(* CODESYS project canbus.20191014.1.project

Project tree, tasks and I/O mapping:
  Changsha_Xiangji_ARM_Cortex_A9_xilinx_zynq7000_linux : Changsha Xiangji-ARM Cortex A9(xilinx zynq7000)-linux, Changsha Xiangji Hiden Technology Co.Ltd, version 3.5.10.40
    application Application
      libraries: VisuDialogs, * (System); CAA Real Time Clock Extern, 3.5.10.0 (CAA Technical Workgroup); CAA Callback Extern, 3.5.11.0 (CAA Technical Workgroup); CAA Can Low Level Imp Extern, 3.5.11.0 (CAA Technical Workgroup); SysMem, 3.5.12.0 (System); CAA SerialCom, 3.5.12.0 (CAA Technical Workgroup); CAA DTUtil Extern, 3.5.12.0 (CAA Technical Workgroup); SysFile, 3.5.9.0 (System); SysTypes2 Interfaces, * (System); CAA Types Extern, 3.5.13.0 (CAA Technical Workgroup); CAA Can Low Level Extern, 3.5.13.0 (CAA Technical Workgroup); CAA Net Base Services, 3.5.13.0 (CAA Technical Workgroup); Standard, 3.5.13.0 (System); CAA File, 3.5.13.40 (CAA Technical Workgroup)
      task VISU_TASK (cyclic, interval 100 ms, priority 31) calls VisuElems.Visu_Prg
      task task_can (cyclic, interval 4 ms, priority 5) calls prg_can0, prg_can1, prg_test_can
      CAN_COMM/
        program prg_can0 [ST]
        function CAN_Send_MSG [ST]
        program prg_can1 [ST]: can1_get_data1, can1_get_data3, can1_get_data2, can1_set_send_buf
        program prg_test_can [ST]
      visualisation main
      funcs/
    SoftMotion General Axis Pool
    IoDrvMIC7001 : IoDrvMIC7001, Cyber-MI, version 18.11.1
        unmapped channels: Ai00@C16, Ai01@C28, Ai02@C17, Ai03@C29, Ai04@C30, Ai05@C19, Ai06@C31, Ai07@C20, Ai08@C18, Ai09@D18, Ai10@D20, Ai11@D31, Ai12@D19, Ai13@D30, Ai14@D29, Ai15@D17, Ai16@D28, Ai17@D16, Ai18-Do00@C25, Ai19-Do01@C24, Ai20-Do02@C13, Ai21-Do03@C01, Ai22-Do04@C03, Ai23-Do05@C04, Ai24-Do06@C05, Ai25-Do07@C06, Ai26-Do08@C08, Ai27-Do09@C09, Ai28-Do10@C10, Ai29-Do11@C11, Ai30-Do12@D34, Ai31-Do13@D35, Ai32-Do14@D23, Ai33-Do15@D12, Ai34-Do16@D10, Ai35-Do17@D09, Ai36-Do18@D08, Ai37-Do19@D07, Ai38-Do20@D05, Ai39-Do21@D04,
          Ai40-Do22@D03, Ai41-Do23@D02, Ai42-Do24@C23, Ai43-Do25@C35, Ai44-Do26@D24, Ai45-Do27@D13, Ai46-Ao00@C22, Ai47-Ao01@D14, Ai48_Pi02, Ai49_Out5V, Ai50_VCC, Ai51_VCC_L, Ai52_VCC_R, Ai53_Pwm-i0, Ai54_Pwm-i1, Ai55_Pwm-i2, Ai56_Pwm-i3, Ai57_CPU-T, Ai58_G-x, Ai59_G-y, Ai60_G-z, Ai61-reserved, Ai62-IO-cntr, Ai63-CDS-cntr, Di00-Ai00@C16, Di01-Ai01@C28, Di02-Ai02@C17, Di03-Ai03@C29, Di04-Ai04@C30, Di05-Ai05@C19, Di06-Ai06@C31, Di07-Ai07@C20, Di08-Ai08@C18, Di09-Ai09@D18, Di10-Ai10@D20, Di11-Ai11@D31, Di12-Ai12@D19, Di13-Ai13@D30, Di14-Ai14@D29, Di15-Ai15@D17,
          Di16-Ai16@D28, Di17-Ai17@D16, Di18-Ai18@C25, Di19-Ai19@C24, Di20-Ai20@C13, Di21-Ai21@C01, Di22-Ai22@C03, Di23-Ai23@C04, Di24-Ai24@C05, Di25-Ai25@C06, Di26-Ai26@C08, Di27-Ai27@C09, Di28-Ai28@C10, Di29-Ai29@C11, Di30-Ai30@D34, Di31-Ai31@D35, Di32-Ai32@D23, Di33-Ai33@D12, Di34-Ai34@D10, Di35-Ai35@D09, Di36-Ai36@D08, Di37-Ai37@D07, Di38-Ai38@D05, Di39-Ai39@D04, Di40-Ai40@D03, Di41-Ai41@D02, Di42-Ai42@C23, Di43-Ai43@C35, Di44-Ai44@D24, Di45-Ai45@D13, Di46-Ai46@C22, Di47-Ai47@D14, Di48-Pi00@C15, Di49-Pi01@C14, Di50-Pi02@D22, Di51-Pi03@D21, Di52-reserved, Di53-reserved, Di54-reserved, Di55-reserved,
          Di56-reserved, Di57-reserved, Di58-reserved, Di59-reserved, Di60-reserved, Di61-reserved, Di62-reserved, Di63-reserved, Pi00-Di48@C15, Pi01-Di49@C14, Pi02-Di50@D22, Pi03-Di51@D21, Do00-Ai18@C25, Do01-Ai19@C24, Do02-Ai20@C13, Do03-Ai21@C01, Do04-Ai22@C03, Do05-Ai23@C04, Do06-Ai24@C05, Do07-Ai25@C06, Do08-Ai26@C08, Do09-Ai27@C09, Do10-Ai28@C10, Do11-Ai29@C11, Do12-Ai30@D34, Do13-Ai31@D35, Do14-Ai32@D23, Do15-Ai33@D12, Do16-Ai34@D10, Do17-Ai35@D09, Do18-Ai36@D08, Do19-Ai37@D07, Do20-Ai38@D05, Do21-Ai39@D04, Do22-Ai40@D03, Do23-Ai41@D02, Do24-Ai42@C23, Do25-Ai43@C35, Do26-Ai44@D24, Do27-Ai45@D13,
          Do28-Pwmi00@C33, Do29-Pwmi01@C34, Do30-Pwmi02@D25, Do31-Pwmi03@D26, PWM00@C25, PWM01@C24, PWM02@C13, PWM03@C01, PWM04@C03, PWM05@C04, PWM06@C05, PWM07@C06, PWM08@C08, PWM09@C09, PWM10@C10, PWM11@C11, PWM12@D34, PWM13@D35, PWM14@D23, PWM15@D12, PWM16@D10, PWM17@D09, PWM18@D08, PWM19@D07, PWM20@D05, PWM21@D04, PWM22@D03, PWM23@D02, PWM24@C23, PWM25@C35, PWM26@D24, PWM27@D13, PWM28-Pwmi00@C33, PWM29-Pwmi01@C34, PWM30-Pwmi02@D25, PWM31-Pwmi03@D26, PWM_I_0@C33, PWM_I_1@C34, PWM_I_2@D25, PWM_I_3@D26,
          Ao00-Ai46@C22, Ao01-Ai47@D14, LED_run, LED_err, LED_usr, ctrl_ai_raw, ctrl_adjust, ctrl_adj0, ctrl_adj1, ctrl_adj2, ctrl_adj3, ctrl_adj4
  5ce3da45-db07-42e7-a21c-a00fff4ed8f6|C:\Users\Administrator\Desktop\robotview1.bmp
  5ce3da45-db07-42e7-a21c-a00fff4ed8f6|C:\Users\Administrator\Desktop\robotview2.bmp
  text list GlobalTextList
  5ce3da45-db07-42e7-a21c-a00fff4ed8f6|C:\Users\Administrator\Desktop\1129.bmp
  5ce3da45-db07-42e7-a21c-a00fff4ed8f6|C:\Users\Administrator\Desktop\robotview0.bmp
*)

// Changsha_Xiangji_ARM_Cortex_A9_xilinx_zynq7000_linux/Application/CAN_COMM/prg_can0
PROGRAM prg_can0   //CAN0   与底盘和显示屏通信
VAR
	hCan0:CAA.HANDLE:=0;
    CanWriteData : ARRAY[0..7] OF BYTE;
    CanWriteMsgID:UDINT;
	CanReadData : ARRAY[0..7] OF BYTE;  
	CanReadMsgID:UDINT;
	bModifyTimeFlag :BOOL := FALSE;
	
	//通过CAN总线从底盘读到的信息
	can_data_ready:BOOL := FALSE;
	can_data_speed:BYTE := 0;
	can_data_soc:BYTE := 0;
	
	//通过CAN总线从显示屏读到的信息
	c00byte0bit0_both_wash_sweep:BOOL := FALSE;
	c00byte0bit1_left_wash_sweep:BOOL := FALSE;
	c00byte0bit2_right_wash_sweep:BOOL := FALSE;
	c00byte0bit3_both_sweep:BOOL := FALSE;
	c00byte0bit4_left_sweep:BOOL := FALSE;
	c00byte0bit5_right_sweep:BOOL := FALSE;
	c00byte0bit6_both_wash:BOOL := FALSE;
	c00byte0bit7_left_wash:BOOL := FALSE;
	
	c00byte1bit0_right_wash:BOOL := FALSE;
	c00byte1bit1_stop_sweep:BOOL := FALSE;
	c00byte1bit2_start_motor:BOOL := FALSE;
	c00byte1bit3_stop_motor:BOOL := FALSE;
	c00byte1bit4_speed_add:BOOL := FALSE;
	c00byte1bit5_speed_dec:BOOL := FALSE;
	c00byte1bit6_normal_speed:BOOL := FALSE;
	c00byte1bit7_high_speed:BOOL := FALSE;
	
	c00byte2bit0_garbage_close:BOOL := FALSE;
	c00byte2bit1_garbage_open:BOOL := FALSE;
	c00byte2bit2_garbage_up:BOOL := FALSE;
	c00byte2bit3_garbage_down:BOOL := FALSE;
	c00byte2bit4_fog_bump:BOOL := FALSE;
	c00byte2bit5_selfclean:BOOL := FALSE;
	c00byte2bit6_wastewater_pump:BOOL := FALSE;
	c00byte2bit7_res :BOOL := FALSE;
	
	c00byte3bit0_sweep_high:BOOL := FALSE;
	c00byte3bit1_sweep_middle:BOOL := FALSE;
	c00byte3bit2_sweep_low:BOOL := FALSE;
	c00byte3bit3_highpress_wash:BOOL := FALSE;
	c00byte3bit4_pointshoot_up:BOOL := FALSE;
	c00byte3bit5_pointshoot_down:BOOL := FALSE;
	c00byte3bit6_pointshoot_left:BOOL := FALSE;
	c00byte3bit7_pointshoot_right:BOOL := FALSE;

	c00byte4bit0_drain_start:BOOL := FALSE;
	c00byte4bit1_drain_auto:BOOL := FALSE;
	c00byte4bit2_drain_manual:BOOL := FALSE;
	c00byte4bit3_left_drain:BOOL := FALSE;
	c00byte4bit4_right_drain:BOOL := FALSE;
	c00byte4bit5_sub_drain:BOOL := FALSE;
	c00byte4bit6_selfclean_drain:BOOL := FALSE;
	c00byte4bit7_spout_drain:BOOL := FALSE;
	
	c00byte6bit0_func_test:BOOL := FALSE;
	c00byte6bit1_change_sweeper:BOOL := FALSE;
	c00byte6bit2_intelligent:BOOL := FALSE;
	c00byte6bit3_cleanly:BOOL := FALSE;
	c00byte6bit4_normal:BOOL := FALSE;
	c00byte6bit5_dirty:BOOL := FALSE;
	
	c01byte0bit3_test_watercooler_pump:BOOL := FALSE;
	c01byte0bit4_test_cooler_fan:BOOL := FALSE;
	
	c01byte1bit0_test_sweeper_middle:BOOL := FALSE;
	c01byte1bit1_test_sweeper_low:BOOL := FALSE;
	c01byte1bit2_test_left_sweeper:BOOL := FALSE;
	c01byte1bit3_test_right_sweeper:BOOL := FALSE;
	c01byte1bit4_test_both_sweeper:BOOL := FALSE;
	c01byte1bit5_test_box_down:BOOL := FALSE;
	c01byte1bit6_test_box_up:BOOL := FALSE;
	c01byte1bit7_test_sucker_down:BOOL := FALSE;
	
	c01byte2bit0_test_sucker_up:BOOL := FALSE;
	c01byte2bit1_test_box_open:BOOL := FALSE;
	c01byte2bit2_test_box_close:BOOL := FALSE;
	
	c01byte2bit6_test_left_sweeper_down:BOOL := FALSE;
	c01byte2bit7_test_left_sweeper_up:BOOL := FALSE;
	
	c01byte3bit0_test_right_sweeper_down:BOOL := FALSE;
	c01byte3bit1_test_right_sweeper_up:BOOL := FALSE;
	c01byte3bit2_test_left_sweeper_out:BOOL := FALSE;
	c01byte3bit3_test_right_sweeper_out:BOOL := FALSE;
	c01byte3bit4_test_left_shooter_out:BOOL := FALSE;
	c01byte3bit5_test_right_shooter_out:BOOL := FALSE;
	c01byte3bit6_test_left_shooter_water:BOOL := FALSE;
	c01byte3bit7_test_right_shooter_water:BOOL := FALSE;
	
	c01byte4bit0_test_sucker_water:BOOL := FALSE;
	c01byte4bit1_test_highpress_wash:BOOL := FALSE;
	c01byte4bit2_test_selfclean:BOOL := FALSE;
	c01byte4bit3_test_highpress_pump_gearin:BOOL := FALSE;
	c01byte4bit4_test_fogpump:BOOL := FALSE;
	
	c01byte5bit2_test_wastewater_pump:BOOL := FALSE;
	c01byte5bit3_test_wastewater_valve:BOOL := FALSE;
	
	c01byte6bit0_test_backup_power:BOOL := FALSE;
	
	c02byte45_speed_change :UINT := 0;
	c02byte67_sub_motor_min_speed:UINT := 0;
	
	c03byte01_normal_speed:UINT := 0;
	c03byte23_high_speed:UINT := 0;
	c03byte45_sweeper_speed:UINT := 0;
	
	c04byte01_highpress_pump_overspeed_warning:UINT := 0;
	c04byte23_highpress_pump_overspeed_stop:UINT := 0;
	c04byte45_sub_motor_max_speed:UINT := 0;
	c04byte67_sub_motor_idle_speed:UINT := 0;
	
	//通过CAN总线发送到显示屏的信息
	s00byte0bit0_res:BOOL := FALSE;
	
	s00byte1bit0_res:BOOL := FALSE;
	s00byte1bit1_wastewater_full:BOOL := FALSE;
	s00byte1bit2_oil_filter_block:BOOL := FALSE;
	s00byte1bit3_oil_low:BOOL := FALSE;
	s00byte1bit4_res:BOOL := FALSE;
	s00byte1bit5_tank_no_water:BOOL := FALSE;
	s00byte1bit6_res:BOOL := FALSE;
	s00byte1bit7_back_error_stop:BOOL := FALSE;
	
	s00byte2bit0_wastewater_full_stop:BOOL := FALSE;
	s00byte2bit1_electronic_power_fault:BOOL := FALSE;
	s00byte2bit2_highpress_pump_overspeed_warning:BOOL := FALSE;
	s00byte2bit3_highpress_pump_overspeed_stop:BOOL := FALSE;
	s00byte2bit4_please_close_test:BOOL := FALSE;
	s00byte2bit5_being_back:BOOL := FALSE;
	s00byte2bit6_please_open_motor:BOOL := FALSE;
	s00byte2bit7_please_open_test:BOOL := FALSE;
	
	s00byte3bit0_air_press_low:BOOL := FALSE;
	s00byte3bit1_back_the_truck:BOOL := FALSE;
	s00byte3bit2_res:BOOL := FALSE;
	s00byte3bit3_highpress_pump_not_gearin:BOOL := FALSE;
	s00byte3bit4_water_valve_not_on:BOOL := FALSE;
	s00byte3bit5_highpress_blow_valve_not_on:BOOL := FALSE;
	s00byte3bit6_highpress_water_valve_not_on:BOOL := FALSE;
	s00byte3bit7_please_open_box_door:BOOL := FALSE;
	
	s00byte4bit0_pump_valve_not_no:BOOL := FALSE;
	s00byte4bit1_pump_press_fault:BOOL := FALSE;
	s00byte4bit2_fault_stop:BOOL := FALSE;
	s00byte4bit3_please_putdown_supporter:BOOL := FALSE;
	
	s00byte4bit6_chassis_can_fault:BOOL := FALSE;
	s00byte4bit7_motordriver_can_fault:BOOL :=FALSE;
	
	s00byte5bit0_sub_wastebox_error:BOOL := FALSE;
	s00byte5bit1_sub1_wastebox_full:BOOL := FALSE;
	s00byte5bit2_sub2_wastebox_full:BOOL := FALSE;
	s00byte5bit3_water_release_valve_not_close:BOOL := FALSE;
	s00byte5bit4_water_release_valve_not_copen:BOOL := FALSE;
	s00byte5bit5_backup_power_on:BOOL := FALSE;
	s00byte5bit6_power_low_20percent:BOOL := FALSE;
	s00byte5bit7_chassis_no_high_voltage:BOOL := FALSE;
	
	s00byte6bit0_get_power_switch:BOOL := FALSE;
	s00byte6bit1_highpress_water_valve_on:BOOL := FALSE;
	s00byte6bit2_box_door_close:BOOL := FALSE;
	s00byte6bit3_highpress_blow_valve_on:BOOL := FALSE;
	s00byte6bit4_air_press_low:BOOL := FALSE;
	s00byte6bit5_wastewater_full:BOOL := FALSE;
	s00byte6bit6_left_supporter_down:BOOL := FALSE;
	s00byte6bit7_right_supporter_down:BOOL := FALSE;
	
	s00byte7bit4_fog_pump_press_ok:BOOL := FALSE;
	s00byte7bit5_oil_level_low:BOOL := FALSE;
	s00byte7bit6_oil_filter_block:BOOL := FALSE;
	
	s01byte0bit0_power_on:BOOL := FALSE;
	s01byte0bit1_back_the_truck:BOOL := FALSE;
	s01byte0bit2_res:BOOL := FALSE;
	s01byte0bit3_cleanwater_low:BOOL := FALSE;
	
	s01byte1bit0_box_down:BOOL := FALSE;
	s01byte1bit1_box_up:BOOL := FALSE;
	s01byte1bit2_sucker_down:BOOL := FALSE;
	s01byte1bit3_sucker_up:BOOL := FALSE;
	s01byte1bit4_boxdoor_close:BOOL := FALSE;
	s01byte1bit5_boxdoor_open:BOOL := FALSE;
	s01byte1bit6_left_sweeper_up:BOOL := FALSE;
	s01byte1bit7_left_sweeper_down:BOOL := FALSE;
	
	s01byte2bit0_right_sweeper_up:BOOL := FALSE;
	s01byte2bit1_right_sweeper_down:BOOL := FALSE;
	s01byte2bit2_cleanwater_high:BOOL := FALSE;
	s01byte2bit3_alterable_box_low:BOOL := FALSE;
	s01byte2bit4_res:BOOL := FALSE;
	
	s01byte3bit3_right_shooter_out:BOOL := FALSE;
	s01byte3bit4_left_shooter_out:BOOL := FALSE;
	s01byte3bit5_waterpump_gearin:BOOL := FALSE;
	s01byte3bit6_left_shooter_water:BOOL := FALSE;
	s01byte3bit7_right_shooter_water:BOOL := FALSE;
	
	s01byte4bit0_sucker_shooter_water:BOOL := FALSE;
	s01byte4bit1_selfclean_shooter_water:BOOL := FALSE;
	s01byte4bit2_high_sub_shooter_water:BOOL := FALSE;
	s01byte4bit3_water_release_valve:BOOL := FALSE;
	s01byte4bit4_oil_release_valve:BOOL := FALSE;
	s01byte4bit5_sweeper_middle_speed:BOOL := FALSE;
	s01byte4bit6_sweeper_low_speed:BOOL := FALSE;
	s01byte4bit7_left_sweeper_back:BOOL := FALSE;
	
	s01byte5bit0_left_sweeper_down:BOOL := FALSE;
	s01byte5bit1_right_sweeper_back:BOOL := FALSE;
	s01byte5bit2_right_sweeper_down:BOOL := FALSE;
	s01byte5bit3_left_all_sweep:BOOL := FALSE;
	s01byte5bit5_right_sweep:BOOL := FALSE;
	
	s01byte6bit0_right_all_sweep:BOOL := FALSE;
	s01byte6bit1_box_down:BOOL := FALSE;
	s01byte6bit2_box_up:BOOL := FALSE;
	s01byte6bit3_sucker_up:BOOL := FALSE;
	s01byte6bit4_sucker_down:BOOL := FALSE;
	s01byte6bit5_boxdoor_close:BOOL := FALSE;
	s01byte6bit6_boxdoor_open:BOOL := FALSE;
	s01byte6bit7_cleanwater_pump:BOOL := FALSE;
	
	s01byte7bit1_cooler_pump_motor:BOOL := FALSE;
	s01byte7bit2_cooler_fan:BOOL := FALSE;
	s01byte7bit3_fog_pump:BOOL := FALSE;
	
	s02byte0bit67_right_shooter_out:BYTE := 0;
	
	s02byte1bit01_left_shooter_out:BYTE := 0;
	s02byte1bit23_waterpump_gearin:BYTE := 0;
	s02byte1bit45_left_shooter_valve_open:BYTE := 0;
	s02byte1bit67_right_shooter_valve_open:BYTE := 0;
	
	s02byte2bit01_sucker_shooter_valve_open:BYTE := 0;
	s02byte2bit23_selfclean_shooter_valve_open:BYTE := 0;
	s02byte2bit45_high_sub_shooter_valve_open:BYTE := 0;
	s02byte2bit67_water_release_valve:BYTE := 0;
	
	s02byte3bit01_oil_release_valve:BYTE := 0;
	s02byte3bit23_sweeper_middle_speed:BYTE := 0;
	s02byte3bit45_sweeper_low_speed:BYTE := 0;
	s02byte3bit67_left_sweeper_back:BYTE := 0;
	
	s02byte4bit01_left_sweeper_down:BYTE := 0;
	s02byte4bit23_right_sweeper_back:BYTE := 0;
	s02byte4bit45_right_sweeper_down:BYTE := 0;
	s02byte4bit67_left_all_sweep:BYTE := 0;
	
	s02byte5bit01_right_sweep:BYTE := 0;
	s02byte5bit23_res:BYTE := 0;
	
	s02byte6bit01_right_all_sweep:BYTE := 0;
	s02byte6bit23_box_down:BYTE := 0;
	s02byte6bit45_box_up:BYTE := 0;
	s02byte6bit67_sucker_up:BYTE := 0;
	
	s02byte7bit01_sucker_down:BYTE := 0;
	s02byte7bit23_boxdoor_close:BYTE := 0;
	s02byte7bit45_boxdoor_open:BYTE := 0;
	s02byte7bit67_cleanwater_pump:BYTE := 0;
	
	s03byte0bit01_res:BYTE := 0;
	s03byte0bit23_water_coller_motor:BYTE := 0;
	s03byte0bit45_cooler_fan:BYTE := 0;
	s03byte0bit67_lowpress_pump:BYTE := 0;
	
	s03byte3bit0_all_wash_sweep:BOOL := FALSE;
	s03byte3bit1_left_wash_sweep:BOOL := FALSE;
	s03byte3bit2_right_wash_sweep:BOOL := FALSE;
	s03byte3bit3_all_sweep:BOOL := FALSE;
	s03byte3bit4_left_sweep:BOOL := FALSE;
	s03byte3bit5_right_sweep:BOOL := FALSE;
	s03byte3bit6_all_wash:BOOL := FALSE;
	s03byte3bit7_left_wash:BOOL := FALSE;
	
	s03byte4bit0_right_wash:BOOL := FALSE;
	s03byte4bit1_stop_sweep:BOOL := FALSE;
	s03byte4bit2_fog_pump:BOOL := FALSE;
	s03byte4bit3_selfclean:BOOL := FALSE;
	s03byte4bit4_boxdoor_close:BOOL := FALSE;
	s03byte4bit5_boxdoor_open:BOOL := FALSE;
	s03byte4bit6_box_up:BOOL := FALSE;
	s03byte4bit7_box_down:BOOL := FALSE;
	
	s03byte5bit0_motor_start:BOOL := FALSE;
	s03byte5bit1_motor_stop:BOOL := FALSE;
	s03byte5bit4_normal_speed:BOOL := FALSE;
	s03byte5bit5_high_speed:BOOL := FALSE;
	s03byte5bit6_sweeper_high_speed:BOOL := FALSE;
	s03byte5bit7_sweeper_middle_spped:BOOL := FALSE;
	
	s03byte6bit0_sweeper_low_speed:BOOL := FALSE;
	s03byte6bit1_highpress_wash:BOOL := FALSE;
	s03byte6bit2_drain_start:BOOL := FALSE;
	s03byte6bit3_drain_auto:BOOL := FALSE;
	s03byte6bit4_drain_manual:BOOL := FALSE;
	s03byte6bit5_drain_left_shooter:BOOL := FALSE;
	s03byte6bit6_drain_right_shooter:BOOL := FALSE;
	s03byte6bit7_sub_drain:BOOL := FALSE;
	
	s03byte7bit0_drain_selfclean:BOOL := FALSE;
	s03byte7bit1_change_sweeper:BOOL := FALSE;
	s03byte7bit2_func_test:BOOL := FALSE;
	s03byte7bit3_intelligent:BOOL := FALSE;
	s03byte7bit4_cleanly:BOOL := FALSE;
	s03byte7bit5_normal:BOOL := FALSE;
	s03byte7bit6_dirty:BOOL := FALSE;
	s03byte7bit7_wastewater_pump:BOOL := FALSE;
	
	s04byte0bit0_point_shoot_up:BOOL := FALSE;
	s04byte0bit1_point_shoot_down:BOOL := FALSE;
	s04byte0bit2_point_shoot_left:BOOL := FALSE;
	s04byte0bit3_point_shoot_right:BOOL := FALSE;
	s04byte0bit4_sucker_shooter_drain:BOOL := FALSE;
	
	s04byte1bit3_test_cooler_motor:BOOL := FALSE;
	s04byte1bit4_test_cooler_fan:BOOL := FALSE;
	s04byte1bit5_test_sweeper_middle:BOOL := FALSE;
	s04byte1bit6_test_sweeper_low:BOOL := FALSE;
	s04byte1bit7_test_left_sweep:BOOL := FALSE;
	
	s04byte2bit0_test_right_sweep:BOOL := FALSE;
	s04byte2bit1_test_all_sweep:BOOL := FALSE;
	s04byte2bit2_test_box_down:BOOL := FALSE;
	s04byte2bit3_test_box_up:BOOL := FALSE;
	s04byte2bit4_test_sucker_down:BOOL := FALSE;
	s04byte2bit5_test_sucker_up:BOOL := FALSE;
	s04byte2bit6_test_boxdoor_open:BOOL := FALSE;
	s04byte2bit7_test_boxdoor_close:BOOL := FALSE;
	
	s04byte3bit0_test_left_sweeper_down:BOOL := FALSE;
	s04byte3bit1_test_left_sweeper_up:BOOL := FALSE;
	s04byte3bit2_test_right_sweeper_down:BOOL := FALSE;
	s04byte3bit3_test_right_sweeper_up:BOOL := FALSE;
	s04byte3bit4_test_left_shooter_out:BOOL := FALSE;
	s04byte3bit5_test_right_shooter_out:BOOL := FALSE;
	s04byte3bit6_test_left_shooter_water:BOOL := FALSE;
	s04byte3bit7_test_right_shooter_water:BOOL := FALSE;
	
	s04byte4bit0_test_sucker_water:BOOL := FALSE;
	s04byte4bit1_test_highpress_wash:BOOL := FALSE;
	s04byte4bit2_test_selfclean:BOOL := FALSE;
	s04byte4bit3_test_highpress_pump_gearin:BOOL := FALSE;
	s04byte4bit4_test_fog_pump:BOOL := FALSE;
	s04byte4bit5_test_left_sweeper_out:BOOL := FALSE;
	s04byte4bit6_test_right_sweeper_out:BOOL := FALSE;
	s04byte4bit7_test_wastewater_pump:BOOL := FALSE;
	
	s04byte5bit0_test_wastewater_valve:BOOL := FALSE;
	s04byte5bit1_test_backup_power:BOOL := FALSE;
	s04byte5bit6_motor_starting:BOOL := FALSE;
	s04byte5bit7_system_running:BOOL := FALSE;
	
	s05byte45_speed_change_value:UINT := 0;
	s05byte67_sub_motor_min_speed:UINT := 0;
	
	s06byte01_normal_speed:UINT := 0;
	s06byte23_high_speed:UINT := 0;
	s06byte45_sweeper_speed:UINT := 0;
	
	s07byte01_highpress_pump_high_speed:UINT := 0;
	s07byte23_highpress_pump_high_speed_stop:UINT := 0;
	s07byte45_sub_motor_max_speed:UINT := 0;
	s07byte67_sub_motor_idle_speed:UINT := 0;
	
	s08byte01_real_torque:UINT := 0;
	s08byte23_real_speed:UINT := 0;
	s08byte45_bus_voltage:UINT := 0;
	s08byte67_phase_current:UINT := 0;
	
	s09byte01_max_dirve_torque:UINT := 0;
	s09byte23_max_brake_torque:UINT := 0;
	s09byte4_temp_controller:BYTE := 0;
	s09byte5_temp_motor:BYTE := 0;
	s09byte67_motor_max_speed:UINT := 0;
	
	s10byte0bit23_direction_cw:BYTE := 0;
	s10byte0bit45_motor_mode:BYTE := 0;
	s10byte0bit67_motor_stat:BYTE := 0;
	
	s10byte1bit01_bus_low_voltage:BYTE := 0;
	s10byte1bit23_bus_high_voltage:BYTE := 0;
	s10byte1bit45_ctrller_high_temp:BYTE := 0;
	s10byte1bit67_motor_high_temp:BYTE := 0;
	
	s10byte2bit01_igbt_fault:BYTE := 0;
	s10byte2bit23_overspeed:BYTE := 0;
	s10byte2bit45_comm_error:BYTE := 0;
	s10byte2bit67_short:BYTE := 0;
	
	s10byte3bit01_motor_overload:BYTE := 0;
	s10byte3bit23_selfcheck_fault:BYTE := 0;
	s10byte3bit45_low_voltage:BYTE := 0;
	s10byte3bit67_sensor_fault:BYTE := 0;
	
	s11byte0_chassis_power_percent:BYTE := 0;
	s11byte1_res :BYTE := 0;
	s11byte23_speed_set_value:UINT := 0;
	s11byte45_version:UINT := 0;
	
	//底盘handle
	hReceiver_ready:CAA.HANDLE;
	hReceiver_speed:CAA.HANDLE;
	hReceiver_soc:CAA.HANDLE;
	
	//显示屏 0x0c00 074f ~ 0x0c04 074f
	hRecver_screen:CAA.HANDLE;
	
	tmp_byte:BYTE;
	tmp_uint:UINT;
	Err:CAA.ERROR;
	
	hMsg : CAA.HANDLE;
	nReceived : CAA.COUNT;
	nAvailable: CAA.COUNT;
	ReadErr   : CAA.ERROR;
	MsgID     : CL2I.COBID;	
	pRxData :POINTER TO CL2I.DATA;
	
	can_stat : DINT := 0;
END_VAR

CASE can_stat OF
	0:   //init can port0 and port1
		hCan0 := cl2.DriverOpenH(usiNetId:=0,uiBaudRate:=250,xSupport29Bits:=TRUE,ctMessages:=100,peError:=ADR(Err));	 //CAN1
		IF hCan0 > 0 THEN
			can_stat := 10;
		END_IF
	
	10: //create receiver for data
		//创建接收底盘信息的接收器: ID:0x18c21726,  byte6.bit2  READY灯	
	  	hReceiver_ready := CL2.CreateMaskReceiver(hDriver := hCan0,
			cobIdValue := 16#18C21726, //cobID value
			cobIdMask := 16#FFFFFFFF, //cobID mask ==> all bits of value are relevant									
			xRTRValue := FALSE, //no RTR messages
			xRTRMask := FALSE, //activate RTR filter ==> xRTRValue will be checked
			x29BitIdValue := TRUE, //29 bit CAN messages
			x29BitIdMask := TRUE, //activate 29 bit filter ==> x29BitIdValue will be checked
			xTransmitValue := FALSE, //only receive messages, no transmit message loopback
			xTransmitMask := FALSE, //activate transmit mask filter ==> xTransmitValue will be checked
			xAlwaysNewest := FALSE, //FALSE := receiver with queue; TRUE: only newest message
			eEvent := CB.EVENT.NO_EVENT,  //no receive event
			xEnableSyncWindow := FALSE, //not implemented
			peError := ADR(Err) //optional pointer to error
			);
		//创建接收底盘信息的接收器: ID:0x18c31726,  byte7  车速	
	  	hReceiver_speed := CL2.CreateMaskReceiver(hDriver := hCan0,
			cobIdValue := 16#18C31726, //cobID value
			cobIdMask := 16#FFFFFFFF, //cobID mask ==> all bits of value are relevant									
			xRTRValue := FALSE, //no RTR messages
			xRTRMask := FALSE, //activate RTR filter ==> xRTRValue will be checked
			x29BitIdValue := TRUE, //29 bit CAN messages
			x29BitIdMask := TRUE, //activate 29 bit filter ==> x29BitIdValue will be checked
			xTransmitValue := FALSE, //only receive messages, no transmit message loopback
			xTransmitMask := FALSE, //activate transmit mask filter ==> xTransmitValue will be checked
			xAlwaysNewest := FALSE, //FALSE := receiver with queue; TRUE: only newest message
			eEvent := CB.EVENT.NO_EVENT, //no receive event
			xEnableSyncWindow := FALSE, //not implemented
			peError := ADR(Err) //optional pointer to error
			);	
		
		//创建接收底盘信息的接收器: ID:0x182126f4,  byte0*0.4  剩余SOC百分比
		hReceiver_soc := CL2.CreateMaskReceiver(hDriver := hCan0,
			cobIdValue := 16#182126F4, //cobID value
			cobIdMask := 16#FFFFFFFF, //cobID mask ==> all bits of value are relevant									
			xRTRValue := FALSE, //no RTR messages
			xRTRMask := FALSE, //activate RTR filter ==> xRTRValue will be checked
			x29BitIdValue := TRUE, //no 29 bit CAN messages
			x29BitIdMask := TRUE, //activate 29 bit filter ==> x29BitIdValue will be checked
			xTransmitValue := FALSE, //only receive messages, no transmit message loopback
			xTransmitMask := FALSE, //activate transmit mask filter ==> xTransmitValue will be checked
			xAlwaysNewest := FALSE, //FALSE := receiver with queue; TRUE: only newest message
			eEvent := CB.EVENT.NO_EVENT, //no receive event
			xEnableSyncWindow := FALSE, //not implemented
			peError := ADR(Err) //optional pointer to error
		);
		//创建接收显示屏信息的接收器: ID:0x0cxx074f
		hRecver_screen := CL2.CreateMaskReceiver(hDriver := hCan0,
			cobIdValue := 16#0C00074F, //cobID value  
			cobIdMask := 16#FFFCFFFF, //cobID mask	0c00074f,0c01074f,0c02074f,0c03074f,							
			xRTRValue := FALSE, //no RTR messages
			xRTRMask := FALSE, //activate RTR filter ==> xRTRValue will be checked
			x29BitIdValue := TRUE, //no 29 bit CAN messages
			x29BitIdMask := TRUE, //activate 29 bit filter ==> x29BitIdValue will be checked
			xTransmitValue := FALSE, //only receive messages, no transmit message loopback
			xTransmitMask := FALSE, //activate transmit mask filter ==> xTransmitValue will be checked
			xAlwaysNewest := FALSE, //FALSE := receiver with queue; TRUE: only newest message
			eEvent := CB.EVENT.NO_EVENT, //no receive event
			xEnableSyncWindow := FALSE, //not implemented
			peError := ADR(Err) //optional pointer to error
		);
		
		IF (hReceiver_ready <> 0 AND hReceiver_speed <> 0 AND hReceiver_soc <> 0 AND hRecver_screen <> 0 ) THEN
			 can_stat := 20;
		ELSE
			RETURN;
		END_IF
	
	20:  //receive data
		//接收底盘信息: ID:0x18c21726,  byte6.bit2  READY灯	
		nReceived := cl2.GetMsgCount(hReceiverId :=hReceiver_ready, peError := ADR(ReadErr));
		IF nReceived <> 0 THEN
			hMsg := cl2.Read(hReceiverId :=hReceiver_ready,pctMsgLeft:=ADR(nAvailable),peError:=ADR(ReadErr));
			pRxData := cl2.GetMessageDataPointer(hMessage:= hMsg,peError:=ADR(ReadErr));	
			tmp_byte := pRxData^[6];
			can_data_ready := tmp_byte.2;
			cl2.FreeMessage(hMsg);
		END_IF

		//接收底盘信息: ID:0x18c31726,  byte7  车速	
		nReceived := cl2.GetMsgCount(hReceiverId :=hReceiver_speed, peError := ADR(ReadErr));
		IF nReceived <> 0 THEN
			hMsg := cl2.Read(hReceiverId :=hReceiver_speed,pctMsgLeft:=ADR(nAvailable),peError:=ADR(ReadErr));
			pRxData := cl2.GetMessageDataPointer(hMessage:= hMsg,peError:=ADR(ReadErr));	
			can_data_speed := pRxData^[6];
			cl2.FreeMessage(hMsg);
		END_IF

		//接收底盘信息: ID:0x182126f4,  byte0*0.4  剩余SOC百分比
		nReceived := cl2.GetMsgCount(hReceiverId :=hReceiver_soc, peError := ADR(ReadErr));
		IF nReceived <> 0 THEN
			hMsg := cl2.Read(hReceiverId :=hReceiver_soc,pctMsgLeft:=ADR(nAvailable),peError:=ADR(ReadErr));
			pRxData := cl2.GetMessageDataPointer(hMessage:= hMsg,peError:=ADR(ReadErr));	
			tmp_uint := ANY_TO_UINT(pRxData^[0]);
			can_data_soc := ANY_TO_BYTE(tmp_uint*2/5);
			cl2.FreeMessage(hMsg);
		END_IF	

		//接收显示屏信息: ID:0x0cXX074f
		nReceived := cl2.GetMsgCount(hReceiverId :=hRecver_screen, peError := ADR(ReadErr));
		IF nReceived <> 0 THEN
			hMsg := cl2.Read(hReceiverId :=hRecver_screen,pctMsgLeft:=ADR(nAvailable),peError:=ADR(ReadErr));
			pRxData := cl2.GetMessageDataPointer(hMessage:= hMsg,peError:=ADR(ReadErr));	
			MsgID := cl2.GetMessageId(hMessage := hMsg, peError := ADR(ReadErr));
			//处理接收数据
			//proc_screen_data(MsgID := MsgID, pRxData := pRxData);
			cl2.FreeMessage(hMsg);
		END_IF
		
		can_stat := 30;
	30:  //send data to screen
		// 12帧数据一起发送，以后可以根据需要调整发送间隔
		
		//填充发送缓冲区
		
		can_stat := 20;

	100:   //error
		
END_CASE

END_PROGRAM

// Changsha_Xiangji_ARM_Cortex_A9_xilinx_zynq7000_linux/Application/CAN_COMM/prg_can1
PROGRAM prg_can1    //CAN1   与上装电机驱动器通信
VAR
	hCan1:CAA.HANDLE:=0;
    CanWriteData : ARRAY[0..7] OF BYTE;
    CanWriteMsgID:UDINT;
	CanReadData : ARRAY[0..7] OF BYTE;  
	CanReadMsgID:UDINT;
	bModifyTimeFlag :BOOL := FALSE;
	
	//通过CAN总线从驱动器读到的信息
	c11byte01_torque:UINT:= 0;
	c11byte23_speed:UINT:= 0;
	c11byte45_voltage:UINT:=0;
	c11byte67_current:UINT:= 0;
	
	c12byte01_drv_torque_max:UINT:= 0;
	c12byte23_brk_torque_max:UINT := 0;
	c12byte4_temp_controller:INT:= 0; //offset:  -40
	c12byte5_temp_motor:INT := 0;  //offset: -40
	c12byte67_speed_max:UINT:= 0;  
	
	c13byte0bit23_cw:BYTE:=0; //00:stop, 01:ccw,  10:cw
	c13byte0bit45_mode:BYTE := 01; //01:drive, 10:brake
	c13byte0bit67_stat:BYTE := 00; //00: enable, 01:running, 10:stop, 11:fault
	
	c13byte1bit01_low_vol:BYTE := 00; //00: normal, 01:warning, 10: fault
	c13byte1bit23_high_vol:BYTE := 0;
	c13byte1bit45_temp_ctrler:BYTE := 0;
	c13byte1bit67_temp_motor:BYTE := 0;
	
	c13byte2bit01_igbt:BYTE := 0;
	c13byte2bit23_speed:BYTE := 0;
	c13byte2bit45_comm:BYTE := 0;
	c13byte2bit67_short:BYTE := 0;
	
	c13byte3bit01_overload:BYTE := 0;
	c13byte3bit23_selfcheck:BYTE := 0;
	c13byte3bit45_low_voltage:BYTE := 0;
	c13byte3bit67_sensor:BYTE := 0;
	
	
	//发送给驱动器的信息
	byte0bit6_enable:BOOL := FALSE;
	byte0bit45_cw:BYTE := 01;  //01:CCW,  10:CW 方向
	byte0bit23_ctrl:BYTE := 01; //01:转矩， 10：转速
	byte0bit01_mode:BYTE := 01;  //01:牵引， 10: 制动
	byte12_torque:UINT:= 0; //转矩
	byte34_speed:UINT := 0;  //转速
	


	hReceiver1:CAA.HANDLE;
	hReceiver2:CAA.HANDLE;
	hReceiver3:CAA.HANDLE;
	tmp_byte:BYTE;
	tmp_uint:UINT;
	Err:CAA.ERROR;
	
	hMsg : CAA.HANDLE;
	nReceived : CAA.COUNT;
	nAvailable: CAA.COUNT;
	ReadErr   : CAA.ERROR;
	MsgID     : CL2I.COBID;	
	pRxData :POINTER TO CL2I.DATA;
	
	can_stat : DINT := 0;
END_VAR

CASE can_stat OF
	0:   //init can port1
		hCan1 := cl2.DriverOpenH(usiNetId:=1,uiBaudRate:=250,xSupport29Bits:=TRUE,ctMessages:=100,peError:=ADR(Err));	 //CAN1
		IF hCan1 > 0 THEN
			can_stat := 10;
		END_IF
	
	10: //create receiver for data
		//接收驱动器信息1: ID:0x0C112AEE,  
	  	hReceiver1 := CL2.CreateMaskReceiver(hDriver := hCan1,
			cobIdValue := 16#0C112AEE, //cobID value
			cobIdMask := 16#FFFFFFFF, //cobID mask ==> all bits of value are relevant									
			xRTRValue := FALSE, //no RTR messages
			xRTRMask := FALSE, //activate RTR filter ==> xRTRValue will be checked
			x29BitIdValue := TRUE, //29 bit CAN messages
			x29BitIdMask := TRUE, //activate 29 bit filter ==> x29BitIdValue will be checked
			xTransmitValue := FALSE, //only receive messages, no transmit message loopback
			xTransmitMask := FALSE, //activate transmit mask filter ==> xTransmitValue will be checked
			xAlwaysNewest := FALSE, //FALSE := receiver with queue; TRUE: only newest message
			eEvent := CB.EVENT.NO_EVENT,  //no receive event
			xEnableSyncWindow := FALSE, //not implemented
			peError := ADR(Err) //optional pointer to error
			);
		//接收驱动器信息2: ID:0x0C122AEE	
	  	hReceiver2 := CL2.CreateMaskReceiver(hDriver := hCan1,
			cobIdValue := 16#0C122AEE, //cobID value
			cobIdMask := 16#FFFFFFFF, //cobID mask ==> all bits of value are relevant									
			xRTRValue := FALSE, //no RTR messages
			xRTRMask := FALSE, //activate RTR filter ==> xRTRValue will be checked
			x29BitIdValue := TRUE, //29 bit CAN messages
			x29BitIdMask := TRUE, //activate 29 bit filter ==> x29BitIdValue will be checked
			xTransmitValue := FALSE, //only receive messages, no transmit message loopback
			xTransmitMask := FALSE, //activate transmit mask filter ==> xTransmitValue will be checked
			xAlwaysNewest := FALSE, //FALSE := receiver with queue; TRUE: only newest message
			eEvent := CB.EVENT.NO_EVENT, //no receive event
			xEnableSyncWindow := FALSE, //not implemented
			peError := ADR(Err) //optional pointer to error
			);	
		
		//接收驱动器信息3: ID:0x0C132AEE
		hReceiver3 := CL2.CreateMaskReceiver(hDriver := hCan1,
			cobIdValue := 16#0C132AEE, //cobID value
			cobIdMask := 16#FFFFFFFF, //cobID mask ==> all bits of value are relevant									
			xRTRValue := FALSE, //no RTR messages
			xRTRMask := FALSE, //activate RTR filter ==> xRTRValue will be checked
			x29BitIdValue := TRUE, //no 29 bit CAN messages
			x29BitIdMask := TRUE, //activate 29 bit filter ==> x29BitIdValue will be checked
			xTransmitValue := FALSE, //only receive messages, no transmit message loopback
			xTransmitMask := FALSE, //activate transmit mask filter ==> xTransmitValue will be checked
			xAlwaysNewest := FALSE, //FALSE := receiver with queue; TRUE: only newest message
			eEvent := CB.EVENT.NO_EVENT, //no receive event
			xEnableSyncWindow := FALSE, //not implemented
			peError := ADR(Err) //optional pointer to error
		);
		IF (hReceiver1 <> 0 AND hReceiver2 <> 0 AND hReceiver3 <> 0 ) THEN
			 can_stat := 20;
		ELSE
			RETURN;
		END_IF
	20:  //send data 
		can1_set_send_buf(ADR(canWriteData));
		CAN_Send_MSG(hCan1, 16#0801EE2A, 8, CanWriteData);
		can_stat := 30;
	
	30:  //receive data
		//接收驱动器信息1: ID:0x0C112AEE,  
		nReceived := cl2.GetMsgCount(hReceiverId :=hReceiver1, peError := ADR(ReadErr));
		IF nReceived <> 0 THEN
			hMsg := cl2.Read(hReceiverId :=hReceiver1,pctMsgLeft:=ADR(nAvailable),peError:=ADR(ReadErr));
			pRxData := cl2.GetMessageDataPointer(hMessage:= hMsg,peError:=ADR(ReadErr));	
			can1_get_data1(pRxData);
			cl2.FreeMessage(hMsg);
		END_IF

		//接收驱动器信息2: ID:0x0C122AEE
		nReceived := cl2.GetMsgCount(hReceiverId :=hReceiver2, peError := ADR(ReadErr));
		IF nReceived <> 0 THEN
			hMsg := cl2.Read(hReceiverId :=hReceiver2,pctMsgLeft:=ADR(nAvailable),peError:=ADR(ReadErr));
			pRxData := cl2.GetMessageDataPointer(hMessage:= hMsg,peError:=ADR(ReadErr));	
			can1_get_data2(pRxData);
			cl2.FreeMessage(hMsg);
		END_IF

		//接收驱动器信息3: ID:0x0C132AEE
		nReceived := cl2.GetMsgCount(hReceiverId :=hReceiver3, peError := ADR(ReadErr));
		IF nReceived <> 0 THEN
			hMsg := cl2.Read(hReceiverId :=hReceiver3,pctMsgLeft:=ADR(nAvailable),peError:=ADR(ReadErr));
			pRxData := cl2.GetMessageDataPointer(hMessage:= hMsg,peError:=ADR(ReadErr));	
			can1_get_data3(pRxData);
			cl2.FreeMessage(hMsg);
		END_IF	
		
		can_stat := 20;
	
	
	100:   //error
		
		
END_CASE

METHOD can1_get_data1 : bool
VAR_INPUT
	pRxData :POINTER TO CL2I.DATA;
END_VAR

VAR
	tmp_byte : BYTE := 0;
	tmp_uint: UINT := 0;
END_VAR
c11byte01_torque := 256*ANY_TO_UINT(pRxData^[1]) + ANY_TO_UINT(pRxData^[0]);
c11byte23_speed :=  256*ANY_TO_UINT(pRxData^[3]) + ANY_TO_UINT(pRxData^[2]);
c11byte45_voltage :=  256*ANY_TO_UINT(pRxData^[5]) + ANY_TO_UINT(pRxData^[4]);
c11byte67_current :=  256*ANY_TO_UINT(pRxData^[7]) + ANY_TO_UINT(pRxData^[6]);

can1_get_data1 := TRUE;
END_METHOD

METHOD can1_get_data3 : bool
VAR_INPUT
	pRxData :POINTER TO CL2I.DATA;
END_VAR

VAR
	tmp_byte : BYTE := 0;
	tmp_uint: UINT := 0;
END_VAR
tmp_byte := pRxData^[0];
c13byte0bit23_cw := ANY_TO_BYTE(tmp_byte.3)*2 + ANY_TO_BYTE(tmp_byte.2);
c13byte0bit45_mode := ANY_TO_BYTE(tmp_byte.5)*2 + ANY_TO_BYTE(tmp_byte.4);
c13byte0bit67_stat := ANY_TO_BYTE(tmp_byte.7)*2 + ANY_TO_BYTE(tmp_byte.6); 

tmp_byte := pRxData^[1];
c13byte1bit01_low_vol := ANY_TO_BYTE(tmp_byte.1)*2 + ANY_TO_BYTE(tmp_byte.0);
c13byte1bit23_high_vol := ANY_TO_BYTE(tmp_byte.3)*2 + ANY_TO_BYTE(tmp_byte.2);
c13byte1bit45_temp_ctrler := ANY_TO_BYTE(tmp_byte.5)*2 + ANY_TO_BYTE(tmp_byte.4);
c13byte1bit67_temp_motor := ANY_TO_BYTE(tmp_byte.7)*2 + ANY_TO_BYTE(tmp_byte.6);

tmp_byte := pRxData^[2];
c13byte2bit01_igbt := ANY_TO_BYTE(tmp_byte.1)*2 + ANY_TO_BYTE(tmp_byte.0);
c13byte2bit23_speed := ANY_TO_BYTE(tmp_byte.3)*2 + ANY_TO_BYTE(tmp_byte.2);
c13byte2bit45_comm := ANY_TO_BYTE(tmp_byte.5)*2 + ANY_TO_BYTE(tmp_byte.4);
c13byte2bit67_short := ANY_TO_BYTE(tmp_byte.7)*2 + ANY_TO_BYTE(tmp_byte.6);

tmp_byte := pRxData^[3];
c13byte3bit01_overload := ANY_TO_BYTE(tmp_byte.1)*2 + ANY_TO_BYTE(tmp_byte.0);
c13byte3bit23_selfcheck := ANY_TO_BYTE(tmp_byte.3)*2 + ANY_TO_BYTE(tmp_byte.2);
c13byte3bit45_low_voltage := ANY_TO_BYTE(tmp_byte.5)*2 + ANY_TO_BYTE(tmp_byte.4);
c13byte3bit67_sensor := ANY_TO_BYTE(tmp_byte.7)*2 + ANY_TO_BYTE(tmp_byte.6);

can1_get_data3 := TRUE;
END_METHOD

METHOD can1_get_data2 : bool
VAR_INPUT
	pRxData :POINTER TO CL2I.DATA;
END_VAR

VAR
	tmp_byte : BYTE := 0;
	tmp_uint: UINT := 0;
END_VAR

c12byte01_drv_torque_max := 256*ANY_TO_UINT(pRxData^[1]) + ANY_TO_UINT(pRxData^[0]);
c12byte23_brk_torque_max := 256*ANY_TO_UINT(pRxData^[3]) + ANY_TO_UINT(pRxData^[2]);
c12byte4_temp_controller := ANY_TO_INT(pRxData^[4]) - 40;
c12byte5_temp_motor := ANY_TO_INT(pRxData^[5]) - 40;
c12byte67_speed_max :=  256*ANY_TO_UINT(pRxData^[7]) + ANY_TO_UINT(pRxData^[6]);

can1_get_data2 := TRUE;
END_METHOD

METHOD can1_set_send_buf : bool
VAR_INPUT
	pData :POINTER TO CL2I.DATA;
END_VAR

VAR
	tmp_byte : BYTE := 0;
END_VAR
tmp_byte := 0;
tmp_byte.6 := byte0bit6_enable;
tmp_byte := tmp_byte + byte0bit45_cw*16;
tmp_byte := tmp_byte + byte0bit23_ctrl*4;
tmp_byte := tmp_byte + byte0bit01_mode*1;

can1_set_send_buf := TRUE;
END_METHOD

END_PROGRAM

// Changsha_Xiangji_ARM_Cortex_A9_xilinx_zynq7000_linux/Application/CAN_COMM/CAN_Send_MSG
FUNCTION CAN_Send_MSG : BOOL
VAR_INPUT
	h:	dword;     //hCan
	TMsgID   : CL2I.COBID;
    TusiLen  : USINT;
	TData    : ARRAY[0..7] OF BYTE;    	
END_VAR
VAR
   Send:CAA.HANDLE;
   WriteErr   : CL2.ERROR;
   p_data:POINTER TO CL2I.DATA;
END_VAR

IF  (0=h) THEN
	RETURN;
END_IF 

Send := cl2.CreateMessage(hDriver := h,
                          cobID := TMsgID,
						  usiLength := TusiLen,
						  xRTR := FALSE,
						  x29BitID := TRUE,
						  peError := ADR(WriteErr));
						  
IF Send <> CAA.gc_hINVALID THEN
	p_data := cl2.GetMessageDataPointer(hMessage := Send,peError:=ADR(WriteErr));
	IF (WriteErr = CL2.ERROR.NO_ERROR) THEN
		SysMemCpy(pDest:=p_data,pSrc:=ADR(TData),udiCount:=SIZEOF(TData));
	END_IF
	
	WriteErr := cl2.Write(hDriver := h,hMessage:=Send,usiPriority:=1,xEnableSyncWindow:=FALSE);
	IF (WriteErr <> CL2.ERROR.NO_ERROR) THEN
        cl2.FreeMessage(hMessage:=Send);		
	END_IF
	
	p_data := CAA.gc_pNULL;
	Send:=CAA.gc_hINVALID;	
END_IF

END_FUNCTION

// Changsha_Xiangji_ARM_Cortex_A9_xilinx_zynq7000_linux/Application/CAN_COMM/prg_test_can
PROGRAM prg_test_can
VAR
	hCan0:CAA.HANDLE:=0;
	hCan1:CAA.HANDLE:=0;
	cmd_test:BOOL := FALSE;
    CanWriteData : ARRAY[0..7] OF BYTE;
    CanWriteMsgID:UDINT;
	CanReadData : ARRAY[0..7] OF BYTE;  
	CanReadMsgID:UDINT;		
	test_01:BOOL := FALSE;
	test_02:BOOL := FALSE;
	test_03:BOOL := FALSE;
	test_04:BOOL := FALSE;
	test_05:BOOL := FALSE;
	test_06:BOOL := FALSE;
	test_07:BOOL := FALSE;
	
END_VAR


IF NOT cmd_test THEN 
	RETURN;
END_IF

hCan0 := prg_can0.hCan0;
hCan1 := prg_can1.hCan1;

IF test_01 THEN
	CanWriteData[0] := 123;
	CanWriteData[1] := 1;
	CanWriteData[6] := 234;
	CAN_Send_MSG(hCan0, 16#0C112AEE, 8, CanWriteData);	
	test_01 := FALSE;
END_IF

IF test_02 THEN
	CAN_Send_MSG(hCan0, 16#0C122AEE, 8, CanWriteData);	
	test_02 := FALSE;
END_IF

IF test_03 THEN
	CAN_Send_MSG(hCan0, 16#0C132AEE, 8, CanWriteData);
	test_03 := FALSE;	
END_IF

IF test_04 THEN
	CAN_Send_MSG(hCan1, 16#18C21726, 8, CanWriteData);
	test_04 := FALSE;	
END_IF

END_PROGRAM

// Changsha_Xiangji_ARM_Cortex_A9_xilinx_zynq7000_linux/Application/main
VISUALIZATION main  // 2x2
END_VISUALIZATION
